// TIA Portal V19 export
DATA_BLOCK "FinalCut"   // DB139
// stored: InstanceOfName FinalCut_FB, InstanceOfType FB
"FinalCut_FB"
   // VAR_INPUT
   //    AreaInterface : "AreaInterface";
   //    ZSI : "udt_ZoneSafetyInterface";
   //    DSI : "udt_DeviceSafetyInterface";
   //    DataIn : Struct
   //       CutHead : "ValveMachine_DataIn";
   //       DrawHead : "ValveMachine_DataIn";
   //       MarkHead : "ValveMachine_DataIn";
   //       Locking : "ValveMachine_DataIn";
   //       Locking_PressureAI : Int;
   //    END_STRUCT;
   //    CIn : Struct
   //       PressureRunning : Bool;
   //       MaterialStandstill : Bool;
   //       EnableCutHead : Bool;
   //       EnableDrawHead : Bool;
   //       EnableMarkHead : Bool;
   //       PPrf_PrgNo : DInt;
   //       CutHead_Manager : "ValveMachine_Manager";
   //       DrawHead_Manager : "ValveMachine_Manager";
   //       MarkHead_Manager : "ValveMachine_Manager";
   //    END_STRUCT;
   //    Config : Struct
   //       CheckRestPosition : Bool;
   //       CutHead : "ValveMachine_Config";
   //       DrawHead : "ValveMachine_Config";
   //       MarkHead : "ValveMachine_Config";
   //       Locking : "ValveMachine_Config";
   //       Locking_AI_HighLimit : Real;
   //       Locking_AI_LowLimit : Real;
   //    END_STRUCT;
   // END_VAR
   // VAR_OUTPUT
   //    MachineInterface : "MachineInterface";
   //    DataOut : Struct
   //       CutHead : "ValveMachine_DataOut";
   //       DrawHead : "ValveMachine_DataOut";
   //       MarkHead : "ValveMachine_DataOut";
   //       Locking : "ValveMachine_DataOut";
   //    END_STRUCT;
   //    COut : Struct
   //       CutHead : "ValveMachine_COut";
   //       DrawHead : "ValveMachine_COut";
   //       MarkHead : "ValveMachine_COut";
   //       Locking : "ValveMachine_COut";
   //       Avg_R_to_W_Time : Time;
   //       Avg_W_to_R_Time : Time;
   //       AllAtRest : Bool;
   //    END_STRUCT;
   // END_VAR
   // VAR_IN_OUT
   //    PersistentValues : "udt_FinalCut_Pers";
   // END_VAR
   // VAR
   //    Sts : Struct
   //       CycleTime : Struct
   //          CutHead : Struct
   //             DT_W_Start : DTL;
   //             DT_W_Stop : DTL;
   //             DT_R_Start : DTL;
   //             DT_R_Stop : DTL;
   //             R_To_W_Exe : Bool;
   //             W_To_R_Exe : Bool;
   //             R_To_W_Items : Int;
   //             R_To_W_Sum : Time;
   //             W_To_R_Items : Int;
   //             W_To_R_Sum : Time;
   //          END_STRUCT;
   //          DrawHead : Struct
   //             DT_W_Start : DTL;
   //             DT_W_Stop : DTL;
   //             DT_R_Start : DTL;
   //             DT_R_Stop : DTL;
   //             R_To_W_Exe : Bool;
   //             W_To_R_Exe : Bool;
   //             R_To_W_Items : Int;
   //             R_To_W_Sum : Time;
   //             W_To_R_Items : Int;
   //             W_To_R_Sum : Time;
   //          END_STRUCT;
   //          MarkHead : Struct
   //             DT_W_Start : DTL;
   //             DT_W_Stop : DTL;
   //             DT_R_Start : DTL;
   //             DT_R_Stop : DTL;
   //             R_To_W_Exe : Bool;
   //             W_To_R_Exe : Bool;
   //             R_To_W_Items : Int;
   //             R_To_W_Sum : Time;
   //             W_To_R_Items : Int;
   //             W_To_R_Sum : Time;
   //          END_STRUCT;
   //          PPrf_PrgNoSave : DInt;
   //       END_STRUCT;
   //       LockingPressure : Real;
   //       WorkPressureOk : Bool;
   //       MinPressureOk : Bool;
   //    END_STRUCT;
   //    Ctrl : Struct
   //       Reload : Struct
   //          CutHead : Bool;
   //          DrawHead : Bool;
   //          MarkHead : Bool;
   //          Locking : Bool;
   //       END_STRUCT;
   //       RstAlarms : Bool;
   //    END_STRUCT;
   //    Alarm : Struct
   //       CutHead : "ValveAlr";
   //       DrawHead : "ValveAlr";
   //       MarkHead : "ValveAlr";
   //       Locking : "ValveAlr";
   //       Locking_NotAWork : Bool;
   //    END_STRUCT;
   //    Warning : Struct
   //       CutHead : "ValveMachine_Wng";
   //       DrawHead : "ValveMachine_Wng";
   //       MarkHead : "ValveMachine_Wng";
   //       Locking : "ValveMachine_Wng";
   //       CutHead_NotAtRest : Bool;
   //       DrawHead_NotAtRest : Bool;
   //       MarkHead_NotAtRest : Bool;
   //       Locking_NotAWork : Bool;
   //       MaterialNotStandstill : Bool;
   //    END_STRUCT;
   //    HMI : Struct
   //       CutHead : Struct
   //          Last_R_to_W_ID : DInt;
   //          Last_R_to_W_Time : Time;
   //          Last_W_to_R_ID : DInt;
   //          Last_W_to_R_Time : Time;
   //          Avg_R_to_W_Time : Time;
   //          Avg_W_to_R_Time : Time;
   //          Buffer_R_to_W_Time : Array[1..10] of Struct
   //             ID : DInt;
   //             Value : Time;
   //          END_STRUCT;
   //          Buffer_W_to_R_Time : Array[1..10] of Struct
   //             ID : DInt;
   //             Value : Time;
   //          END_STRUCT;
   //       END_STRUCT;
   //       DrawHead : Struct
   //          Last_R_to_W_ID : DInt;
   //          Last_R_to_W_Time : Time;
   //          Last_W_to_R_ID : DInt;
   //          Last_W_to_R_Time : Time;
   //          Avg_R_to_W_Time : Time;
   //          Avg_W_to_R_Time : Time;
   //          Buffer_R_to_W_Time : Array[1..10] of Struct
   //             ID : DInt;
   //             Value : Time;
   //          END_STRUCT;
   //          Buffer_W_to_R_Time : Array[1..10] of Struct
   //             ID : DInt;
   //             Value : Time;
   //          END_STRUCT;
   //       END_STRUCT;
   //       MarkHead : Struct
   //          Last_R_to_W_ID : DInt;
   //          Last_R_to_W_Time : Time;
   //          Last_W_to_R_ID : DInt;
   //          Last_W_to_R_Time : Time;
   //          Avg_R_to_W_Time : Time;
   //          Avg_W_to_R_Time : Time;
   //          Buffer_R_to_W_Time : Array[1..10] of Struct
   //             ID : DInt;
   //             Value : Time;
   //          END_STRUCT;
   //          Buffer_W_to_R_Time : Array[1..10] of Struct
   //             ID : DInt;
   //             Value : Time;
   //          END_STRUCT;
   //       END_STRUCT;
   //    END_STRUCT;
   //    CutHead : "ValveMachine_FB";
   //    DrawHead : "ValveMachine_FB";
   //    MarkHead : "ValveMachine_FB";
   //    Locking : "ValveMachine_FB";
   //    TON_CutHead_Pause : IEC_TIMER;
   //    TON_CutHead_Duration : IEC_TIMER;
   //    TON_DrawHead_Pause : IEC_TIMER;
   //    TON_DrawHead_Duration : IEC_TIMER;
   //    TON_MarkHead_Pause : IEC_TIMER;
   //    TON_MarkHead_Duration : IEC_TIMER;
   //    TON_LockingTimeOut : IEC_TIMER;
   //    PE_Aux : Struct
   //       CutHead : Struct
   //          AtRest : Bool;
   //          AtWork : Bool;
   //          NotAtRest : Bool;
   //          NotAtWork : Bool;
   //       END_STRUCT;
   //       DrawHead : Struct
   //          AtRest : Bool;
   //          AtWork : Bool;
   //          NotAtRest : Bool;
   //          NotAtWork : Bool;
   //       END_STRUCT;
   //       MarkHead : Struct
   //          AtRest : Bool;
   //          AtWork : Bool;
   //          NotAtRest : Bool;
   //          NotAtWork : Bool;
   //       END_STRUCT;
   //    END_STRUCT;
   //    i : Int;
   // END_VAR
BEGIN
END_DATA_BLOCK
